TYPE TYP_VAC_GEN_HW_OUT :
STRUCT
	EnableVac AT %Q* : BOOL;
	ReleaseVac AT %Q* : BOOL;
END_STRUCT
END_TYPE

(* stored: Version 1.1.0.1, ProductVersion 3.1.4024.12
   DUT TYP_VAC_GEN_HW_OUT: Id {4e293fc1-0893-4764-a299-a1dcd7ffc441} *)
